// TIA Portal V20 export
TYPE "typeCmHmiInterfaceSoftCam"
// stored: Access Published, Namespace Unit1.Em3
   STRUCT
      topTapeAxisX : "Unit1.Em3.typeCmHmiInterfaceSoftCamtopTapeAxisX";
      topTapeAxisY : "Unit1.Em3.typeCmHmiInterfaceSoftCamtopTapeAxisY";
   END_STRUCT;
END_TYPE
